TYPE ST_System_KKKW_Zustand :
STRUCT
	Betrieb_Anford			: BOOL;
	Betrieb_Soll				: BOOL;
	Betrieb					: BOOL;

	Regelung_Sollw			: REAL;
	Regelung_Modus				: SINT;

	Freigabe					: BOOL;
	Freigabe_Deakt			: BOOL;
	Freigabe_Code			: WORD;

	Stoerung					: BOOL;
	Stoerung_Code			: WORD;

	Warnung					: BOOL;
	Warnung_Code			: WORD;

	Status					: SINT;
	Status_Vorl				: BOOL;
	Status_Nachl				: BOOL;

	Status_Vorl_Stellventil	: BOOL;
	Status_Vorl_Pumpen		: BOOL;
	Status_Nachl_Stellventil: BOOL;
	Status_Nachl_Pumpen		: BOOL;
	Status_Wiedereinschalten: BOOL;

	Quittierung				: BOOL;

END_STRUCT
END_TYPE

(* stored: Version 1.1.0.1, ProductVersion 3.1.4024.9
   DUT ST_System_KKKW_Zustand: Id {923e4589-caab-4401-9bd3-d2a427f39b57} *)
